TYPE ST_HMI_Monitor_switchgear :
STRUCT
	//Switchgear
	b_ACDetectedBusbar			: BOOL;
	b_ACDetectedInput			: BOOL;
	b_DCDetected				: BOOL;
	b_PeNeutralLink				: BOOL;
	b_ACInputState				: BOOL; //summary of MCCB and contactor state.
	b_InputSync					: BOOL;
	r_ACInputPower				: REAL;
	b_NetContactorState			: BOOL; //summary of netcontactor left and right close state.
	b_ACOutputState				: BOOL;
	r_ACOutputPower				: REAL; 
	b_DCCouplingState			: BOOL;
	r_DCCouplingCurrent			: REAL;
END_STRUCT
END_TYPE

(* stored: Version 1.1.0.1, ProductVersion 3.1.4026.18
   DUT ST_HMI_Monitor_switchgear: Id {59c826a0-6123-4cfb-bf3c-e5de94218bb0} *)
